// TwinCAT 3 PLC project P1
// ProgramVersion: 3.1.4024.0
// libraries:
//   Tc2_Standard, * (Beckhoff Automation GmbH)
//   Tc2_System, * (Beckhoff Automation GmbH)
//   Tc3_Module, * (Beckhoff Automation GmbH)
// project tree:
//   / GlobalTextList.TcGTLO, PlcTask.TcTTO, Visualization Manager.TcVMO (not stored), Visualization.TcVIS
//   POUs/ FB_Add.TcPOU, MAIN.TcPOU
// real-time tasks:
//   TASK PlcTask: cycle T#10ms, priority 20, ADS port 350

CONFIGURATION P1
    RESOURCE PLC ON TwinCAT3
        TASK PlcTask(INTERVAL := T#10ms, PRIORITY := 20);
        PROGRAM MAIN WITH PlcTask : MAIN;
    END_RESOURCE
END_CONFIGURATION

// ---- POUs/MAIN.TcPOU
PROGRAM MAIN
VAR
	iA: INT;
	iB: INT;
	iC: INT;
	
	fb_add1: FB_Add;
END_VAR

 fb_add1(iIn1:= iA, iIn2:= iB, iOut=> iC);

END_PROGRAM

// ---- POUs/FB_Add.TcPOU
FUNCTION_BLOCK FB_Add
VAR_INPUT	
	iIn1,iIn2: INT;
END_VAR
VAR_OUTPUT
	iOut: INT;
END_VAR
VAR
END_VAR

 iOut := iIn1+iIn2;

END_FUNCTION_BLOCK

// ---- Visualization.TcVIS
VISUALIZATION Visualization  // 2x2
END_VISUALIZATION
